ABB RobotStudio station: MATERIALHANDLING001-05-03-2024.rsstn

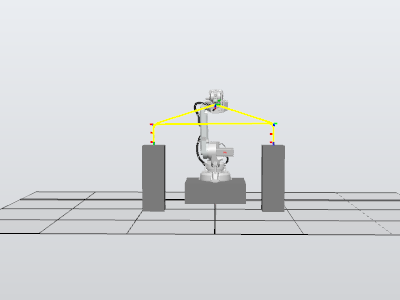
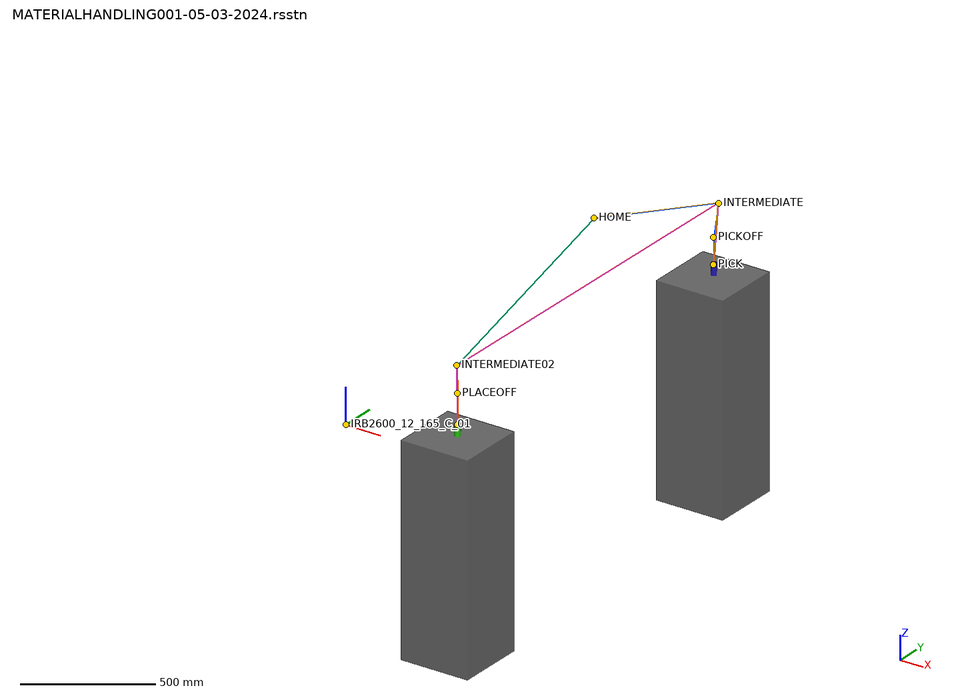
[picture v1: parts stored in the station drawn from their meshes, with robot base, taught points and paths (robot models come from the ABB library and are not in the file)]
Station Station (saved by RobotStudio 22.3.10141.1)
Controller Controller27, task T_ROB1: task frame (RAPID world) sits at (0, 0, 300) mm in the station
Controller Controller27
  mechanical unit ROB_1: IRB2600_12_165_C_01, 6 joints, base frame (0, 0, 0) mm
Layout (positions relative to the parent item):
  - IRB2600_12_165_C_01 [mechanism, from %ABB.RobotStudio.Models.IRB2600%\IRB2600_12_165_C_01.rslib] at (0, 0, 300) mm; joint values [0, 0, 0, 0, 0.5236, 0] (rad or m)
  - concrete [part, from Libraries\concrete.rslib] at (-450, -450, 0) mm
  - SmartComponent_3 [smart component] at (1018.61, 0, 1517.5) mm, rotated rx 180 ry 60 rz 180 deg
      signals: DI Attach
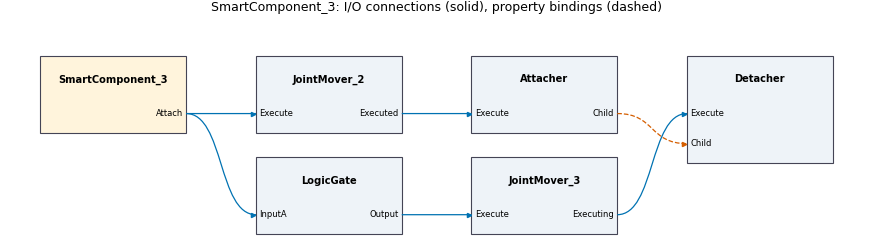
      connections:
        SmartComponent_3.Attach -> JointMover_2.Execute
        JointMover_2.Executed -> Attacher.Execute
        SmartComponent_3.Attach -> LogicGate.InputA
        LogicGate.Output -> JointMover_3.Execute
        JointMover_3.Executing -> Detacher.Execute
        Attacher.Child => Detacher.Child
    - Smart_Gripper_Servo_Fingers [mechanism, from Tools\ABB_Smart_Gripper_Servo_Fingers.rslib] at (0, 0, 0) mm; joint values [0.025] (rad or m)
    - JointMover_2 [smart component, from Components\JointMover.rslib]
        properties: Mechanism=Smart_Gripper_Servo_Fingers; Relative=false; Duration=0; J1=0.023
    - JointMover_3 [smart component, from Components\JointMover.rslib]
        properties: Mechanism=Smart_Gripper_Servo_Fingers; Relative=false; Duration=0; J1=0.025
    - Attacher [smart component, from Components\Attacher.rslib]
        properties: Parent=Smart_Gripper_Servo_Fingers; Flange=0; Child=Part_6; Mount=false; Offset=[0 0 0]; Orientation=[0 0 0]
    - Detacher [smart component, from Components\Detacher.rslib]
        properties: Child=Part_6; KeepPosition=true
    - LogicGate [smart component, from Components\LogicGate.rslib]
        properties: Operator=NOT; Delay=0
  - Tab le01 [part] at (945.63, 643.43, 0) mm, size 300 x 300 x 900 mm
  - Tab le02 [part] at (945.63, -997.26, 0) mm, size 300 x 300 x 900 mm
  - Part_6 [part] at (1095.63, 800, 901.86) mm, size 24 x 23.9 x 50 mm
  - Part_7 [part] at (1095.63, -847.26, 900) mm, size 24 x 23.9 x 50 mm
Attachment: SmartComponent_3 is attached to IRB2600_12_165_C_01 / Link6
Station logic (signal -> signal, property => property):
  Controller27.ATTACH -> SmartComponent_3.Attach
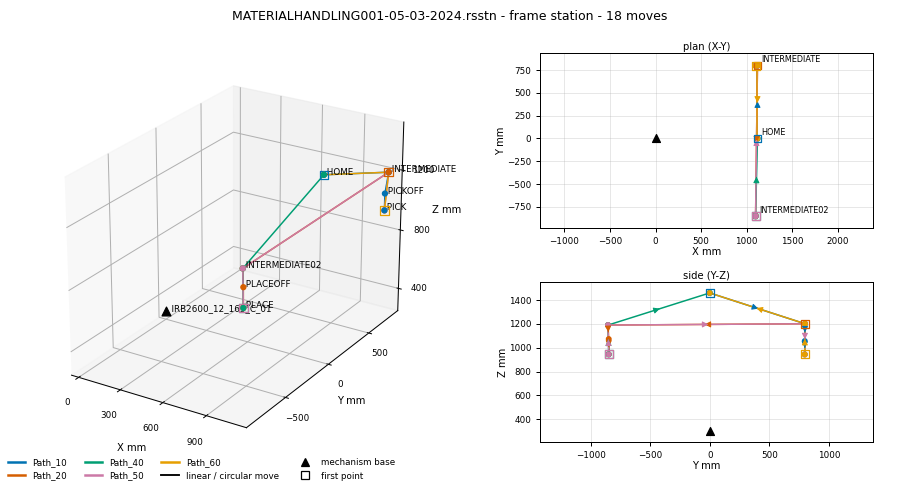
[picture p0: tool path of MATERIALHANDLING001-05-03-2024.rsstn in frame station, 18 of 18 moves have a stored position in this frame; points joined in program order, loops and branches not executed]
Targets, tools, work objects and paths stored in the station, written as RAPID:
! task T_ROB1
MODULE CalibData
  PERS tooldata Servo:=[TRUE,[[0,0,114.2],[1,0,0,0]],[0.215,[8.7,12.3,49.2],[1,0,0,0],0.00021,0.00024,0.00009]];
ENDMODULE

! task T_ROB1
MODULE Module1
  CONST robtarget HOME:=[[1117.512260434,0,1160.4],[0.5,0,0.866025404,0],[-1,0,-1,0],[9E+09,9E+09,9E+09,9E+09,9E+09,9E+09]];
  CONST robtarget INTERMEDIATE:=[[1117.511967148,799.815120038,901.784618895],[0.500000013,-0.000000054,0.866025396,-0.000000006],[0,-1,0,0],[9E+09,9E+09,9E+09,9E+09,9E+09,9E+09]];
  CONST robtarget PICK:=[[1096.652039529,797.809095672,644.214031732],[0.011068168,0.668205625,-0.743241048,-0.031168604],[0,0,-1,0],[9E+09,9E+09,9E+09,9E+09,9E+09,9E+09]];
  CONST robtarget PICKOFF:=[[1096.652039696,797.809100241,756.532496106],[0.011068173,0.668205635,-0.743241039,-0.031168614],[0,0,-1,0],[9E+09,9E+09,9E+09,9E+09,9E+09,9E+09]];
  CONST robtarget INTERMEDIATE02:=[[1096.65204019,-853.574979991,890.67417019],[0.011068219,0.66820569,-0.743240989,-0.031168619],[-1,-1,-2,0],[9E+09,9E+09,9E+09,9E+09,9E+09,9E+09]];
  CONST robtarget PLACE:=[[1096.652032472,-847.399163225,645.087208766],[0.011068277,0.668205662,-0.743241013,-0.031168621],[-1,-1,-2,0],[9E+09,9E+09,9E+09,9E+09,9E+09,9E+09]];
  CONST robtarget PLACEOFF:=[[1096.652025081,-847.399140459,773.429803594],[0.01106825,0.668205653,-0.74324102,-0.031168658],[-1,-1,-2,0],[9E+09,9E+09,9E+09,9E+09,9E+09,9E+09]];
  PROC Path_10()
    MoveL HOME,v1000,z100,Servo\WObj:=wobj0;
    MoveL INTERMEDIATE,v1000,z100,Servo\WObj:=wobj0;
    MoveL PICKOFF,v1000,z100,Servo\WObj:=wobj0;
    MoveL PICK,v1000,z100,Servo\WObj:=wobj0;
    WaitTime 1;
    SetDO ATTACH,1;
    WaitTime 1;
  ENDPROC
  PROC Path_20()
    MoveL INTERMEDIATE,v1000,z100,Servo\WObj:=wobj0;
    MoveL INTERMEDIATE02,v1000,z100,Servo\WObj:=wobj0;
    MoveL PLACEOFF,v1000,z100,Servo\WObj:=wobj0;
    MoveL PLACE,v1000,z100,Servo\WObj:=wobj0;
    WaitTime 1;
    SetDO ATTACH,0;
    WaitTime 1;
  ENDPROC
  PROC Path_30()
    Path_10;
    Path_20;
    Path_40;
    Path_50;
    Path_60;
  ENDPROC
  PROC Path_40()
    MoveL PLACE,v1000,z100,Servo\WObj:=wobj0;
    MoveL INTERMEDIATE02,v1000,z100,Servo\WObj:=wobj0;
    MoveL HOME,v1000,z100,Servo\WObj:=wobj0;
  ENDPROC
  PROC Path_50()
    MoveL PLACE,v1000,z100,Servo\WObj:=wobj0;
    WaitTime 1;
    SetDO ATTACH,1;
    WaitTime 1;
    MoveL INTERMEDIATE02,v1000,z100,Servo\WObj:=wobj0;
    MoveL INTERMEDIATE,v1000,z100,Servo\WObj:=wobj0;
    MoveL PICK,v1000,z100,Servo\WObj:=wobj0;
    WaitTime 1;
    SetDO ATTACH,0;
    WaitTime 1;
  ENDPROC
  PROC Path_60()
    MoveL PICK,v1000,z100,Servo\WObj:=wobj0;
    MoveL INTERMEDIATE,v1000,z100,Servo\WObj:=wobj0;
    MoveL HOME,v1000,z100,Servo\WObj:=wobj0;
  ENDPROC
ENDMODULE

